RoboDK station: Station_test.rdk

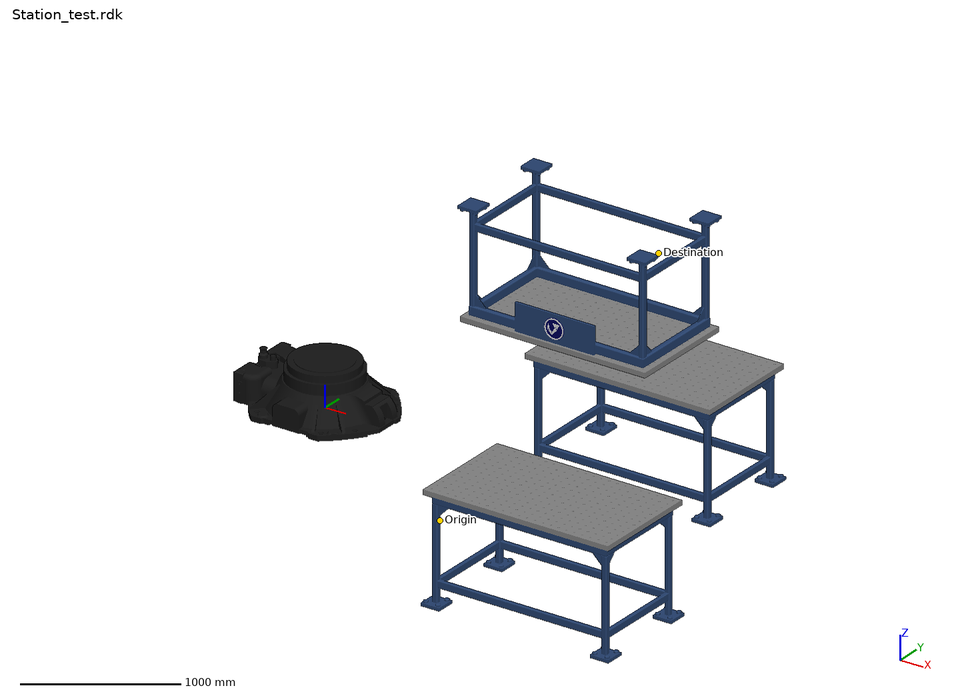
[picture v0: the station drawn from its stored meshes, robots at their saved joint values, targets as dots, program paths as lines]
Station Station_test (saved by RoboDK 5.9.2). Poses are relative to the parent item; angles as X-Y-Z fixed-axis rotations.
  - frame Fanuc M-900iB/700 Base at (0, 1000, 940) mm
    - robot Fanuc M-900iB/700: 6 axes, payload 700 kg, reach 2832 mm, repeatability 0.3 mm, weight 2800 kg
        joint limits [-180, -44, -65, -360, -122, -360] to [180, 110, 95, 360, 122, 360]; home [0, 0, 0, 0, 0, 0]; saved at [-30.964, 14.975, -47.689, 0, -42.311, 30.964]
    - target Origin (Cartesian target) at (1500, -900, 0) mm, rotated rx -180 ry 0 rz 0 deg; joints [-30.964, 14.975, -47.689, 0, -42.311, 30.964] of Fanuc M-900iB/700
    - target Destination (Cartesian target) at (1618.63, 1294.45, 1000) mm, rotated rx -180 ry 0 rz 0 deg; joints [38.65, 19.652, -0.212, 0, -89.788, -38.65] of Fanuc M-900iB/700
    - object Table 1400x800x800mm at (1500, -200, 0) mm, size 1420 x 820 x 800 mm, geometry from Table-1400x800x800mm.sld
    - object Table 1400x800x800mm at (1500, 200, 1000) mm, rotated rx 180 ry 0 rz 0 deg, size 1420 x 820 x 800 mm, geometry from Table-1400x800x800mm.sld
    - object Table 1400x800x800mm at (1500, 900, 500) mm, size 1420 x 820 x 800 mm, geometry from Table-1400x800x800mm.sld
